TYPE ST_AxisRecipe :
	STRUCT
		Velocity		: INT;
		Acceleration	: INT;
		Deceleration	: INT;
	//	Speed			: INT;
		MaxVelocity		: INT;
	END_STRUCT
END_TYPE

(* stored: Version 1.1.0.1, ProductVersion 3.1.4024.15
   DUT ST_AxisRecipe: Id {6aa5ebe1-e8fd-41c7-85ad-1d86b0808233} *)
